(* IEC 61131-3 sources: plc_generation_empirical_study/datasets/task_bank_v0_3_1/tasks/C04_B11_composite, 2 files *)

(* ---- interface.st ---- *)
FUNCTION_BLOCK C04_B11_composite
VAR_INPUT
    A_Signal : BOOL;
    A_Arm : BOOL;
    B_Button : BOOL;
    B_Enable : BOOL;
    B_Reset : BOOL;
    SubsystemBEnable : BOOL;
    CrossReset : BOOL;
END_VAR
VAR_OUTPUT
    A_Pulse : BOOL;
    A_Armed : BOOL;
    B_State : BOOL;
    B_AcceptedPulse : BOOL;
    CrossReady : BOOL;
    CrossBlocked : BOOL;
END_VAR
END_FUNCTION_BLOCK

(* ---- reference.st ---- *)
FUNCTION_BLOCK C04_B11_composite
VAR_INPUT
    A_Signal : BOOL;
    A_Arm : BOOL;
    B_Button : BOOL;
    B_Enable : BOOL;
    B_Reset : BOOL;
    SubsystemBEnable : BOOL;
    CrossReset : BOOL;
END_VAR
VAR_OUTPUT
    A_Pulse : BOOL;
    A_Armed : BOOL;
    B_State : BOOL;
    B_AcceptedPulse : BOOL;
    CrossReady : BOOL;
    CrossBlocked : BOOL;
END_VAR
VAR
    A_PrevSignal : BOOL := FALSE;
    B_PrevButton : BOOL := FALSE;
END_VAR

A_Pulse := A_Arm AND (NOT A_Signal) AND A_PrevSignal;
A_Armed := A_Arm;
A_PrevSignal := A_Signal;

IF CrossReset THEN
    CrossReady := FALSE;
ELSIF A_Pulse THEN
    CrossReady := TRUE;
END_IF;
CrossBlocked := SubsystemBEnable AND (NOT CrossReady);

IF SubsystemBEnable AND CrossReady THEN
    B_AcceptedPulse := FALSE;
    IF B_Reset THEN
        B_State := FALSE;
    ELSIF B_Enable AND B_Button AND (NOT B_PrevButton) THEN
        B_State := NOT B_State;
        B_AcceptedPulse := TRUE;
    END_IF;
    B_PrevButton := B_Button;
ELSE
    B_State := FALSE;
    B_AcceptedPulse := FALSE;
END_IF;

END_FUNCTION_BLOCK
